Staubli VAL3: remMovSphAxis.pgx

program remMovSphAxis(string& sArgs[] (dimensions=1), string& sReturn[] (dimensions=1))
  local bool bOk
  local num nAzi
  local num nEle
  local num nIndex
  local num nRad
  local num nVal
  local string sAxis
  local string sVal
begin
  // Move to a designated point along an axis in
  // spherical coordinates, keeping other axes constant.
  //
  // arguments are "AXIS POS", e.g. "RAD 1000"
  //
  logMsg("call remMovSphAxis")
  //parse args, expecting axis label and a number.
  //We already know we have exactly 2 args.
  nIndex=find(sArgs," ")
  sAxis=left(sArgs,nIndex)
  sVal=delete(sArgs,nIndex+1,0)
  toNum(sVal,nVal,bOk)
  if bOk
    call remCalcHereSph()
    nAzi=nAzHere
    nEle=nElHere
    nRad=nRHere
    switch sAxis
      case "AZI"
        nAzi=nVal
      break
      case "ELE"
        nEle=nVal
      break
      case "RAD"
        nRad=nVal
      break
      default
        call remErrInvalid("MOVSPHAXIS",sAxis,sReturn)
        return
      break
    endSwitch
    call remMovSph(nAzi,nEle,nRad,sReturn)
  else
    call remErrNum("MOVSPHAXIS",sVal,sReturn)
  endIf
end
